INTERFACE ITF_BaseLoggerElement_HMI_Connector EXTENDS
		ITF_BaseLoggerElement_HMI_Connector_Command, ITF_BaseLoggerElement_HMI_Connector_View

END_INTERFACE

(* stored: Version 1.1.0.1
   Itf ITF_BaseLoggerElement_HMI_Connector: Id {4c8dc41f-6fbe-0df0-315f-37d7e9df42d0} *)
